FUNCTION_BLOCK "GCS7_E_MYRA_MDEx"	// FB 36
TITLE = MYRA
//
//COPYRIGHT:    (C) 1996 BY  BUHLER LTD.
//                           CH-9240 UZWIL  SWITZERLAND
//
//PRODUCT:      GCS7
//
//TITLE:        MYRA, MYAG, MDEF / MDEA or MDEE 
//              (OPTO22 or 24V signal) 
//
//REVISION:     GCPROVB 11
//-------------------------------------------------------------------------
//
//IDENT:        AUTHOR:             DEPT:                       DATE:
//
//FB36.5.2      A. Egli             CT3                         07-Mar-2007
//              Update Version 5.1 from G. Shingler CDDP
//              - Addition of command 'N' to allow current values to be read
//              - Addition of command 'b' for MYRA to allow current flowrates
//                to be read
//              - Read of average flowrates removed (command 'm')
//FB36.5.1      A. Egli             CT3                         16-Jan-2007
//              - Read average of ingredient 1 to 7 (command i)
//FB36.5.0      G. Shingler         CDDP                        19-Dec-2006
//              - Read actual weights and actual flowrates for feeders
//              - Correction for log alarms
//FB36.4.10     A. Egli             CT3                         25-Sep-2006
//              - Only send commands to the mills that are connected
//FB36.4.9      Ph. Engler          GP92                        03-May-2006
//              - CmdFaultReset set with Gr.CmdFaultReset (M 12.3)
//FB36.4.8      Ph. Engler          GP92                        28-Apr-2006
//              - MDEF: Send 's' only after a 'D'
//              - MDEF: Only one recipe change at the time
//FB36.4.7      A. Egli             CT3                         22-Dec-2004
//              Command 'S': check also MYRA.OutStatus.Suspended
//FB36.4.6      A. Egli             CT3                         05-Nov-2004
//              New transition StFault --> StOn
//FB36.4.5      A. Egli             CT3                         11-Okt-2004
//              Fault reset when InNoMonLC=1
//FB36.4.4      P.Engler            MU664                       20-Sep-2004
//              Condtion for StWaitForResponse --> StOff
//FB36.4.3      A. Egli             CT3                         17-Jun-2004
//              InNoMonLC:No alarm only warning when InpFaultLC
//FB36.4.2      K. Tischer          CT3                         13-JAN-2004
//              Revision=10
//FB36.4.1      A. Egli             CT3                         11-Nov-2002
//              Compare ParAlarmResetTime <0
//FB36.4.0      A. Egli             CT3                         30-Okt-2002
//              Read Actual values of ingredients
//FB36.3.0      A. Egli             CT3                         17-Jun-2002
//              New Release with one block
//              OPTO22 communication to MYRA,MAG and MDEF 
//FB36.2A       A. Egli             CT3                         04-Mai-1998
//              StFault = StCode 32
//FB36.1A       A. Egli             AEE61                       29-Okt-1997
//              1st Release in S7
//
//-------------------------------------------------------------------------
//
//PURPOSE:      MANUAL : see [MYRxxMAN]
//
//              (*1): LC is connected to PC
//                    PLC used 24V signal as interface to PC 
//                   
//                    NOTE: In case of OPTO22 the signal are internal used 
//
//              (*2): LC is connected to PLC by opto22
//
//
//RESTRICTIONS: S7
//              CmdOff, CmdOn: always active unless local mode
//
//-------------------------------------------------------------------------
//=======================================================
//Log Message: 
//------------------------------------------------------
// 0   Off
// 1   On 
// 9   fault cancelled
//10   fault equipement          
//11   fault fault tolerance
//12   fault fault transmision
//
//15   Communcation Fault Opto22
//16   MYAG Alarm
//
//21   MYRA Alarm Hardware
//22   MYRA Alarm Product 
//23   MYRA Alarm Recipe change
//24   MYRA Alarm Feeder 1
//25   MYRA Alarm Feeder 2
//26   MYRA Alarm Feeder 3
//27   MYRA Alarm Feeder 4
//
//41   MDEF Alarm mill 1  
//42   MDEF Alarm mill 2
//43   MDEF Alarm mill 3
//44   MDEF Alarm mill 4
//
//51   MDEF Wrong recipe 1  
//52   MDEF Wrong recipe 2
//53   MDEF Wrong recipe 3  
//54   MDEF Wrong recipe 4  
//
//
//=======================================================
//StCode:  State               
//------------------------------------------------------
//32  StFault                   
// 1  StOff                     
//41  StOff.HWStop                     StOff + InHWStop
//51  StOff.DPFault                    StOff + InDPFault
// 2  StWaitForResponse         
// 3  StOn.Ok                   
// 4  StOn.Warning              
// 5  StCtoFault                
//
AUTHOR : GS
FAMILY : GCS7LL
NAME : MYRA_MDE
VERSION : 5.2
VAR
  StCode : INT ;	//Element state code
  InEnable : BOOL ;	//Enable to run the element
  InDefReady : BOOL ;	//(*1) Answer from PLC: Recipe to sent to MYRA
  InDefFault : BOOL ;	//(*1) Answer from PC:  not eble to send recipe to MYRA
  InNoMonLC : BOOL ;	//No alarm only warning when InpFaultLC
  CmdNewValue : BOOL ;	//Send new target values: Send Flowrate to MYRA
  CmdNewJob : BOOL ;	//Send RecipeNr and Job-Nr to MYRA
  InpOutOfTolerance : BOOL ;	//(*1) Digital input 1=Fault
  InpFaultLc : BOOL ;	//(*1) Digital input 1=HW fault of MYRA
  CmdOff : BOOL ;	//Pulse to stop the element immediately (manual mode)
  CmdOn : BOOL ;	//Pulse to start the element immediately (manual mode)
  CmdNext : BOOL ;	//Pulse to start the element in automatic mode (see global flags)
  CmdFaultReset : BOOL ;	//Command to reset fault
  InLocal : BOOL ;	//1= Local mode (no fault by start with service switch)
  InManual : BOOL ;	//1= Manual/ 0=Automatic
  InReport : BOOL ;	//Report of all state transitions
  spare0307 : BOOL ;
  InHWStop : BOOL ;	//HW stop is detected, no fault
  InDPFault : BOOL ;	//DP-Fault is detected, no fault
  OutWarning : BOOL ;	//Out of tolerance, ParDelayWarning end
  OutDefRequested : BOOL ;	//Definition requested : PC must send recipe to MYRA
  OutComFault : BOOL ;	//Communication vault OPTO22
  OutEnabled : BOOL ;	//Enable to run MYRA (internal used)
  OutpAlarmReset : BOOL ;	//(*1) Digital output: Trigger for alarm reset
  OutpRelease : BOOL ;	//(*1) Digital output: Release measuring
  StOff : BOOL ;	//Element is stopped
  StWaitForResponse : BOOL ;	//PC must send new recipe to MYRA
  StOn : BOOL ;
  StCtoFault : BOOL ;
  StFault : BOOL ;
  MDEF1 : STRUCT 	//OPTO22: MDEF1
   CmdNewRecipe : BOOL ;	//Send recipe to mill
   CmdAlarmReset : BOOL ;	//Send to Mill
   OutSendRecipeNrActive : BOOL ;	//Send of recipe nr is active
   OutSendRecipeNrDone : BOOL ;	//RecipeNr is sent
   OutWrongRecipe : BOOL ;	//Status 4, 6 or 10
   OutAlarm : BOOL ;	//Command 'a'
   StNotOK : BOOL ;
   StOK : BOOL ;
   StFault : BOOL ;
   InRecipeNr : INT ;	//Command 'D'
   Status : INT ;	//Command 's'
  END_STRUCT ;
  MDEF2 : STRUCT 	//OPTO22: MDEF2
   CmdNewRecipe : BOOL ;	//Send recipe to mill
   CmdAlarmReset : BOOL ;	//Send to Mill
   OutSendRecipeNrActive : BOOL ;	//Send of recipe nr is active
   OutSendRecipeNrDone : BOOL ;	//RecipeNr is sent
   OutWrongRecipe : BOOL ;	//Status 4, 6 or 10
   OutAlarm : BOOL ;	//Command 'a'
   StNotOK : BOOL ;
   StOK : BOOL ;
   StFault : BOOL ;
   InRecipeNr : INT ;	//Command 'D'
   Status : INT ;	//Command 's'
  END_STRUCT ;
  MDEF3 : STRUCT 	//OPTO22: MDEF3
   CmdNewRecipe : BOOL ;	//Send recipe to mill
   CmdAlarmReset : BOOL ;	//Send to Mill
   OutSendRecipeNrActive : BOOL ;	//Send of recipe nr is active
   OutSendRecipeNrDone : BOOL ;	//RecipeNr is sent
   OutWrongRecipe : BOOL ;	//Status 4, 6 or 10
   OutAlarm : BOOL ;	//Command 'a'
   StNotOK : BOOL ;
   StOK : BOOL ;
   StFault : BOOL ;
   InRecipeNr : INT ;	//Command 'D'
   Status : INT ;	//Command 's'
  END_STRUCT ;
  MDEF4 : STRUCT 	//OPTO22: MDEF4
   CmdNewRecipe : BOOL ;	//Send recipe to mill
   CmdAlarmReset : BOOL ;	//Send to Mill
   OutSendRecipeNrActive : BOOL ;	//Send of recipe nr is active
   OutSendRecipeNrDone : BOOL ;	//RecipeNr is sent
   OutWrongRecipe : BOOL ;	//Status 4, 6 or 10
   OutAlarm : BOOL ;	//Command 'a'
   StNotOK : BOOL ;
   StOK : BOOL ;
   StFault : BOOL ;
   InRecipeNr : INT ;	//Command 'D'
   Status : INT ;	//Command 's'
  END_STRUCT ;
  MYRA : STRUCT 	//OPTO22: MYRA
   InRecipeNr : INT ;	//Command 'P'
   InJobNr : DINT ;	//Command 'P'
   InFlowrate : DINT ;	//Command 'Q' [kg/h]
   Command : STRUCT 	//Command 'S'
    CheckLimit : BOOL ;
    spare11 : BOOL ;
    spare12 : BOOL ;
    spare13 : BOOL ;
    AlarmReset : BOOL ;	//Is programmed by ASW
    Start : BOOL ;
    spare22 : BOOL ;
    spare23 : BOOL ;
   END_STRUCT ;
   OutAlarm : STRUCT 	//Command 'a'
    SumFault : BOOL ;
    AlarmMYRAHardware : BOOL ;
    AlarmProduct : BOOL ;
    AlarmRecipeChange : BOOL ;
    AlarmFeeder1 : BOOL ;
    AlarmFeeder2 : BOOL ;
    AlarmFeeder3 : BOOL ;
    AlarmFeeder4 : BOOL ;
   END_STRUCT ;
   OutStatus : STRUCT 	//Command 's'
    Started : BOOL ;
    Suspended : BOOL ;
    Remote : BOOL ;
    BatchMode : BOOL ;
    spare4_0 : BOOL ;
    spare4_1 : BOOL ;
    spare4_2 : BOOL ;
    spare4_3 : BOOL ;
    EnableFeeder1 : BOOL ;
    EnableFeeder2 : BOOL ;
    EnableFeeder3 : BOOL ;
    EnableFeeder4 : BOOL ;
    LimitFeeder1 : BOOL ;
    LimitFeeder2 : BOOL ;
    LimitFeeder3 : BOOL ;
    LimitFeeder4 : BOOL ;
   END_STRUCT ;
   OutIngr1 : INT ;	//[1/100%] (Command 'f')
   OutIngr2 : INT ;	//[1/100%] (Command 'f')
   OutIngr3 : INT ;	//[1/100%] (Command 'f')
   OutIngr4 : INT ;	//[1/100%] (Command 'f')
   OutIngr5 : INT ;	//[1/100%] (Command 'f')
   OutIngr6 : INT ;	//[1/100%] (Command 'f')
   OutIngr7 : INT ;	//[1/100%] (Command 'f')
   OutFeeder1Weight : DINT ;	//[5.0] [kg] (Command 'm')
   OutFeeder1Flowrate : DINT ;	//[5.0] [kg/h] (Command 'b')
   OutFeeder2Weight : DINT ;	//[5.0] [kg] (Command 'm')
   OutFeeder2Flowrate : DINT ;	//[5.0] [kg/h] (Command 'b')
   OutFeeder3Weight : DINT ;	//[5.0] [kg] (Command 'm')
   OutFeeder3Flowrate : DINT ;	//[5.0] [kg/h] (Command 'b')
   OutFeeder4Weight : DINT ;	//[5.0] [kg] (Command 'm')
   OutFeeder4Flowrate : DINT ;	//[5.0] [kg/h] (Command 'b')
   OutIngr1Average : INT ;	//[1/100%] (Command 'i')
   OutIngr2Average : INT ;	//[1/100%] (Command 'i')
   OutIngr3Average : INT ;	//[1/100%] (Command 'i')
   OutIngr4Average : INT ;	//[1/100%] (Command 'i')
   OutIngr5Average : INT ;	//[1/100%] (Command 'i')
   OutIngr6Average : INT ;	//[1/100%] (Command 'i')
   OutIngr7Average : INT ;	//[1/100%] (Command 'i')
  END_STRUCT ;
  MYAG : STRUCT 	//OPTO22: MYRG
   Start : BOOL ;	//Command 'I': Is sent to LC (internal used)
   RecipeChange : BOOL ;	//Command 'I': Is sent to LC
   InRecipeNr : INT ;	//ASW: Command 'I': Is sent to LC
   InJobNr : DINT ;	//ASW: Command 'I': Is sent to LC
   OutSumFault : BOOL ;	//Command 'b': Is read from LC
   OutRecipeNr : INT ;	//Command 'b': Is read from LC
   OutJobNr : DINT ;	//Command 'b': Is read from LC
   OutYield1 : INT ;	//Command 'b': Is read from LC
   OutYield2 : INT ;	//Command 'b': Is read from LC
   OutFlowrateAc : DINT ;	//Command 'b': Is read from LC
  END_STRUCT ;
  OutMsg : STRUCT 	//Active Message
   A10LC : BOOL ;
   A11Tolerance : BOOL ;
   A12CommunicationPC : BOOL ;
   A15CommunicationLC : BOOL ;
   A21MYRAHardware : BOOL ;
   A22MYRAProduct : BOOL ;
   A23MYRARecipeChange : BOOL ;
   A24MYRAFeeder1 : BOOL ;
   A25MYRAFeeder2 : BOOL ;
   A26MYRAFeeder3 : BOOL ;
   A27MYRAFeeder4 : BOOL ;
   A41Mill1 : BOOL ;
   A42Mill2 : BOOL ;
   A43Mill3 : BOOL ;
   A44Mill4 : BOOL ;
   A51RecipeMill1 : BOOL ;
   A52RecipeMill3 : BOOL ;
   A53RecipeMill2 : BOOL ;
   A54RecipeMill4 : BOOL ;
  END_STRUCT ;
  OutAlarmNrLog : INT ;	//Last textnumber send to log
  Par : STRUCT
   ParObjectNo : INT ;	//Is used for communication with PC, e.g. for message
   ParMsgType : INT ;	//Is used for message (translation of state)
   ParHornCode : INT ;	//not used
   ParLogOff : BOOL ;	//Report is off
   ParMDEx : BOOL ;	//MDEx: No Delay time if out of tolerance
   ParMYRA : BOOL ;	//OPTO22: MYRA
   ParMDEF : BOOL ;	//OPTO22: MDEF
   ParMYAG : BOOL ;	//OPTO22: MYAG
   ParComDB : INT ;	//OPTO22: Communication DB
   ParLCIdx : INT ;	//OPTO22: Index of data record
   ParLCAddr : INT ;	//OPTO22: Address of LC
   ParNoOfMDEF : INT ;	//OPTO22: Number of connected MDEF
   ParDelayFault : INT ;	//Delay time, until the element changes to fault
   ParAlarmResetTime : INT ;	//Pulse length for OutpFaultReset
   ParResponseTime : INT ;	//Maximum time to wait for answer from PC
   ParDelayWarning : INT ;	//Delay time, until the element changes to StWarning
   OutDelayTime : INT ;	//Actual time
   spare24 : INT ;
   OutHelpFlags : STRUCT 	//Internal used
    OutFaultResetDone : BOOL ;
    OutTestNewAlarm : BOOL ;
    CmdNewValue : BOOL ;
    CmdNewJob : BOOL ;
    OutAlarmActive : BOOL ;
    FlagCheckLimit : BOOL ;
   END_STRUCT ;
   OutComFlags : STRUCT
    a_rDone : BOOL ;
    s_rDone : BOOL ;
    k_Done : BOOL ;
    b_Done : BOOL ;
    D_Done : BOOL ;
    A_Done : BOOL ;
    P_Done : BOOL ;
    Q_Done : BOOL ;
    S_Done : BOOL ;
    I_Done : BOOL ;
    f_rDone : BOOL ;
    m_Done : BOOL ;	//[5.0]
    i_rDone : BOOL ;	//[5.1]
    N_Done : BOOL ;	//[5.2]
   END_STRUCT ;
   OutMillNr : INT ;	//Used for MDEF Telegram
  END_STRUCT ;
END_VAR
VAR_TEMP
  tmpLOGvalue : WORD ;	//LOG value
  tmpLenDyn : DINT ;
  tmpReport : BOOL ;	//Global LOG all
  tmpEnable : BOOL ;	//Global enable
  tmpLocal : BOOL ;
  tmpTimeDone : BOOL ;
  tmpLocalFault : BOOL ;
  tmpOpto22 : BOOL ;
  tmpFBNO : INT ;	//Number of the actual FB
  tmpCommand : INT ;
  tmpComDB : INT ;
  tmpReturn : INT ;
  tmpFault : BOOL ;
  tmpWrongRecipe : BOOL ;
  tmpAddrMsg : DWORD ;
  tmpPar : STRUCT
   ParObjectNo : INT ;	//Is used for communication with PC, e.g. for message
   ParMsgType : INT ;	//Is used for message (translation of state)
   ParHornCode : INT ;	//not used
   ParLogOff : BOOL ;	//Report is off
   ParMDEx : BOOL ;	//MDEx: No Delay time if out of tolerance
   ParMYRA : BOOL ;	//OPTO22: MYRA
   ParMDEF : BOOL ;	//OPTO22: MDEF
   ParMYAG : BOOL ;	//OPTO22: MYAG
   ParComDB : INT ;	//OPTO22: Communication DB
   ParLCIdx : INT ;	//OPTO22: Index of data record
   ParLCAddr : INT ;	//OPTO22: Address of LC
   ParNoOfMDEF : INT ;	//OPTO22: Number of connected MDEF
   ParDelayFault : INT ;	//Delay time, until the element changes to fault
   ParAlarmResetTime : INT ;	//Pulse length for OutpFaultReset
   ParResponseTime : INT ;	//Maximum time to wait for answer from PC
   ParDelayWarning : INT ;	//Delay time, until the element changes to StWarning
   OutMillNr : INT ;	//Used for MDEF Telegram
  END_STRUCT ;
  tmpReturn1 : INT ;
END_VAR
BEGIN
NETWORK
TITLE =  Start Global
      L     170;
      T     #tmpLenDyn;	//--> Len dynamic data in byte
      L     #Par.ParComDB;
      T     #tmpComDB;
      L     36;
      T     #tmpFBNO;
      A     #Par.ParMYRA;
      O     #Par.ParMDEF;
      O     #Par.ParMYAG;
      =     #tmpOpto22;
      TAR2;
      L     DW#16#FFFFFF;
      AD;
      L     P##OutMsg;
      +D;
      T     #tmpAddrMsg;
NETWORK
TITLE =  Call back function (***Opto22***)
////*************************************************
////***             O P T O 22                    ***
////*************************************************
//
//This functions are called by FBxxx (COM) 
      AN    #tmpOpto22;
      JC    PC;
      OPN   DB [#tmpComDB];
      L     0;
      L     DBW 32;	//COM.Element.CODE;
      ==I;
      JC    PC;
//Check if object has moved
      L     #Par.ParObjectNo;
      L     DBD 60;	//COM.LC0.AddrPara;       
      ==D;
      JC    COok;
      BEC;
//=============================================
COok: L     DBB 76;	//COM.Telegram.Command;
      T     #tmpCommand;
      L     1;
      L     DBW 32;	//COM.Element.CODE;
      ==I;
      JC    Send;
      L     2;
      ==I;
      JC    Rcv;
      L     4;	//NAK
      L     DBW 32;	//COM.Element.CODE;
      ==I;
      S     #OutComFault;	//fault MYEB communication
      BEU;
//===== Prepare data for send =================================
//Read telegram length
Send: L     #tmpCommand;
      L     'a';
      ==I;
      AN    #Par.ParMYRA;
      L     4;	//Lenght in byte
      JC    Sndx;
      L     #tmpCommand;
      L     'a';
      ==I;
      A     #Par.ParMYRA;
      L     2;	//Lenght in byte
      JC    Sndx;
      L     #tmpCommand;	//[4.0]
      L     'f';	//[4.0]
      ==I;	//[4.0]
      A     #Par.ParMYRA;	//[4.0]
      L     35;	//Lenght in byte             //[4.0]
      JC    Sndx;
      L     #tmpCommand;	//[5.1]
      L     'i';	//[5.1]
      ==I;	//[5.1]
      A     #Par.ParMYRA;	//[5.1]
      L     28;	//Lenght in byte             //[5.1]
      JC    Sndx;
      L     #tmpCommand;	//[5.0]
      L     'm';	//[5.0]
      ==I;	//[5.0]
      A     #Par.ParMYRA;	//[5.0]
      L     64;	//Lenght in byte //[5.0]
      JC    Sndx;	//[5.0]
      L     #tmpCommand;
      L     's';
      ==I;
      AN    #Par.ParMYRA;
      L     2;	//Lenght in byte
      JC    Sndx;
      L     #tmpCommand;
      L     's';
      ==I;
      A     #Par.ParMYRA;
      L     3;	//Lenght in byte
      JC    Sndx;
      L     #tmpCommand;
      L     'b';	//MYAG
      ==I;
      L     25;	//Lenght in byte
      A     #Par.ParMYAG;	//[5.2]
      JC    Sndx;
      L     #tmpCommand;	//[5.2]
      L     'b';	//[5.2] MYRA
      ==I;	//[5.2]
      L     69;	//[5.2] Lenght in byte
      A     #Par.ParMYRA;	//[5.2]
      JC    Sndx;	//[5.2]
      JU    SndA;
Sndx: T     DBW 86;	//COM.Telegram.LenAnswer
      BEU;
//--------------------
//Send A [3.0]
//--------------------
SndA: L     #tmpCommand;
      L     'A';
      <>I;
      JC    SndD;
// command 1
      L     0;
      T     DBW 40;	//COM.Element.AddrOffset
      L     #Par.OutMillNr;
      T     DBD 36;	//COM.Element.InOutValue
      L     11;	//Convert DInt to 1-ASCII
      T     DBW 0;	//COM.CODE
      CDB;	//ComDB->Instanz-DB
      UC    "GCS7_RS485Ctrl";	//Convert (CODE=DBW0)
      CDB;	//ElementDB->Instanz-DB
      L     1;	//Lenght in byte
      T     DBW 78;	//COM.Telegram.Len
      L     0;	//Lenght in byte
      T     DBW 86;	//COM.Telegram.LenAnswer
      BEU;
//--------------------------
//Send D
//--------------------------
SndD: NOP   0;
      L     #tmpCommand;
      L     'D';
      <>I;
      JC    SndI;
      L     0;	//Character offset
      T     DBW 40;	//COM.Element.AddrOffset
      L     1;
      L     #Par.OutMillNr;
      ==I;
      L     #MDEF1.InRecipeNr;
      JC    SD1;
      L     2;
      L     #Par.OutMillNr;
      ==I;
      L     #MDEF2.InRecipeNr;
      JC    SD1;
      L     3;
      L     #Par.OutMillNr;
      ==I;
      L     #MDEF3.InRecipeNr;
      JC    SD1;
      L     #MDEF4.InRecipeNr;
SD1:  T     DBD 36;	//COM.Element.InOutValue
      L     13;	//Convert DInt to 3-ASCII
      T     DBW 0;	//COM.CODE
      CDB;	//ComDB->Instanz-DB
      UC    "GCS7_RS485Ctrl";	//Convert (CODE=DBW0)
      CDB;	//ElementDB->Instanz-DB
      L     3;	//Lenght in byte
      T     DBW 78;	//COM.Telegram.Len
      L     0;	//Lenght in byte
      T     DBW 86;	//COM.Telegram.LenAnswer
      BEU;
//--------------------------
//Send I
//--------------------------
SndI: NOP   0;
      L     #tmpCommand;
      L     'I';
      <>I;
//[5.2]      JC    SndP
      JC    SndN;	//[5.2]
//Start
      L     0;	//Character offset
      T     DBW 40;	//COM.Element.AddrOffset
      L     0;
      T     DBD 36;	//COM.Element.InOutValue
      A     #MYAG.Start;
      =     DBX 39.0;
      L     11;	//Convert DInt to 1-ASCII
      T     DBW 0;	//COM.CODE
      CDB;	//ComDB->Instanz-DB
      UC    "GCS7_RS485Ctrl";	//Convert (CODE=DBW0)
      CDB;	//ElementDB->Instanz-DB
//Recipe change
      L     1;	//Character offset
      T     DBW 40;	//COM.Element.AddrOffset
      L     0;
      T     DBD 36;	//COM.Element.InOutValue
      A     #InManual;
      ON    #InLocal;
      AN    #InDefReady;
      =     #MYAG.RecipeChange;
      =     DBX 39.0;
      L     11;	//Convert DInt to 1-ASCII
      T     DBW 0;	//COM.CODE
      CDB;	//ComDB->Instanz-DB
      UC    "GCS7_RS485Ctrl";	//Convert (CODE=DBW0)
      CDB;	//ElementDB->Instanz-DB
//RecipeNr
      L     2;	//Character offset
      T     DBW 40;	//COM.Element.AddrOffset
      L     #MYAG.InRecipeNr;
      T     DBD 36;	//COM.Element.InOutValue
      L     12;	//Convert DInt to 1-ASCII
      T     DBW 0;	//COM.CODE
      CDB;	//ComDB->Instanz-DB
      UC    "GCS7_RS485Ctrl";	//Convert (CODE=DBW0)
      CDB;	//ElementDB->Instanz-DB
//JobNr
      L     4;	//Character offset
      T     DBW 40;	//COM.Element.AddrOffset
      L     #MYAG.InJobNr;
      T     DBD 36;	//COM.Element.InOutValue
      T     DBD 36;	//COM.Element.InOutValue
      L     16;	//Convert DInt to 1-ASCII
      T     DBW 0;	//COM.CODE
      CDB;	//ComDB->Instanz-DB
      UC    "GCS7_RS485Ctrl";	//Convert (CODE=DBW0)
      CDB;	//ElementDB->Instanz-DB
      L     10;	//Lenght in byte
      T     DBW 78;	//COM.Telegram.Len
      L     0;	//Lenght in byte
      T     DBW 86;	//COM.Telegram.LenAnswer
      BEU;
//[5.2]--------------------------
//[5.2]Send N
//[5.2]--------------------------
SndN: L     #tmpCommand;	//[5.2]
      L     'N';	//[5.2]
      <>I;	//[5.2]
      JC    SndP;	//[5.2]
//[5.2] Job reference 
      L     0;	//[5.2]Character offset
      T     DBW 40;	//[5.2]COM.Element.AddrOffset
      L     0;	//[5.2]0 =  current job
      T     DBD 36;	//[5.2]COM.Element.InOutValue
      L     16;	//[5.2]Convert DInt to 6-ASCII
      T     DBW 0;	//[5.2]COM.CODE
      CDB;	//[5.2]ComDB->Instanz-DB
      UC    "GCS7_RS485Ctrl";	//[5.2]Convert (CODE=DBW0)
      CDB;	//[5.2]ElementDB->Instanz-DB
      L     6;	//[5.2]Lenght in byte
      T     DBW 78;	//[5.2]COM.Telegram.Len
      L     0;	//[5.2]Lenght in byte
      T     DBW 86;	//[5.2]COM.Telegram.LenAnswer
      BEU;
//--------------------------
//Send P
//--------------------------
SndP: L     #tmpCommand;
      L     'P';
      <>I;
      JC    SndQ;
//RecipeNr 
      L     0;	//Character offset
      T     DBW 40;	//COM.Element.AddrOffset
      L     #MYRA.InRecipeNr;
      T     DBD 36;	//COM.Element.InOutValue
      L     13;	//Convert DInt to 3-ASCII
      T     DBW 0;	//COM.CODE
      CDB;	//ComDB->Instanz-DB
      UC    "GCS7_RS485Ctrl";	//Convert (CODE=DBW0)
      CDB;	//ElementDB->Instanz-DB
//Order Number
      L     3;	//Character offset
      T     DBW 40;	//COM.Element.AddrOffset
      L     #MYRA.InJobNr;
      T     DBD 36;	//COM.Element.InOutValue
      L     16;	//Convert DInt to 6-ASCII
      T     DBW 0;	//COM.CODE
      CDB;	//ComDB->Instanz-DB
      UC    "GCS7_RS485Ctrl";	//Convert (CODE=DBW0)
      CDB;	//ElementDB->Instanz-DB
      L     9;	//Lenght in byte
      T     DBW 78;	//COM.Telegram.Len
      L     0;	//Lenght in byte
      T     DBW 86;	//COM.Telegram.LenAnswer
      BEU;
//--------------------------
//Send Q
//--------------------------
SndQ: L     #tmpCommand;
      L     'Q';
      <>I;
      JC    SndS;
//Flowrate
      L     0;	//Character offset
      T     DBW 40;	//COM.Element.AddrOffset
      L     #MYRA.InFlowrate;
      T     DBD 36;	//COM.Element.InOutValue
      L     16;	//Convert DInt to 6-ASCII
      T     DBW 0;	//COM.CODE
      CDB;	//ComDB->Instanz-DB
      UC    "GCS7_RS485Ctrl";	//Convert (CODE=DBW0)
      CDB;	//ElementDB->Instanz-DB
      L     6;	//Lenght in byte
      T     DBW 78;	//COM.Telegram.Len
      L     0;	//Lenght in byte
      T     DBW 86;	//COM.Telegram.LenAnswer
      BEU;
//--------------------------
//Send S
//--------------------------
SndS: L     #tmpCommand;
      L     'S';
      <>I;
      JC    SndZ;
      A     #MYRA.Command.AlarmReset;
      S     #Par.OutHelpFlags.OutFaultResetDone;
//Start
      L     0;	//Character offset
      T     DBW 40;	//COM.Element.AddrOffset
      L     0;
      T     DBD 36;	//COM.Element.InOutValue
      CALL  "SIEMENS_BLKMOV" (
           SRCBLK                   := #MYRA.Command,
           RET_VAL                  := #tmpReturn,
           DSTBLK                   := DBB 39);
      L     32;	//Convert Hex to 2-ASCII
      T     DBW 0;	//COM.CODE
      CDB;	//ComDB->Instanz-DB
      UC    "GCS7_RS485Ctrl";	//Convert (CODE=DBW0)
      CDB;	//ElementDB->Instanz-DB
      L     2;	//Lenght in byte
      T     DBW 78;	//COM.Telegram.Len
      L     0;	//Lenght in byte
      T     DBW 86;	//COM.Telegram.LenAnswer
      BEU;
SndZ: BEU;
//--- Get done ---------------
//Copy reveived data to element
//--------------------------
//Receive f [4.]
//--------------------------
Rcv:  R     #OutComFault;
      L     #tmpCommand;
      L     'f';
      <>I;
      JC    Rcvi;
//OutIngr1 
      L     0;	//Character offset
      T     DBW 40;	//COM.Element.AddrOffset
      L     25;	//Convert 5-ASCII to DInt
      T     DBW 0;	//COM.CODE
      CDB;	//ComDB->Instanz-DB
      UC    "GCS7_RS485Ctrl";	//Convert (CODE=DBW0)
      CDB;	//ElementDB->Instanz-DB
      L     DBD 36;	//COM.Element.InOutValue
      DTR;
      L     1.000001e-01;
      *R;
      RND;
      T     #MYRA.OutIngr1;
//OutIngr2
      L     5;	//Character offset
      T     DBW 40;	//COM.Element.AddrOffset
      L     25;	//Convert 5-ASCII to DInt
      T     DBW 0;	//COM.CODE
      CDB;	//ComDB->Instanz-DB
      UC    "GCS7_RS485Ctrl";	//Convert (CODE=DBW0)
      CDB;	//ElementDB->Instanz-DB
      L     DBD 36;	//COM.Element.InOutValue
      DTR;
      L     1.000001e-01;
      *R;
      RND;
      T     #MYRA.OutIngr2;
//OutIngr3
      L     10;	//Character offset
      T     DBW 40;	//COM.Element.AddrOffset
      L     25;	//Convert 5-ASCII to DInt
      T     DBW 0;	//COM.CODE
      CDB;	//ComDB->Instanz-DB
      UC    "GCS7_RS485Ctrl";	//Convert (CODE=DBW0)
      CDB;	//ElementDB->Instanz-DB
      L     DBD 36;	//COM.Element.InOutValue
      DTR;
      L     1.000001e-01;
      *R;
      RND;
      T     #MYRA.OutIngr3;
//OutIngr4
      L     15;	//Character offset
      T     DBW 40;	//COM.Element.AddrOffset
      L     25;	//Convert 5-ASCII to DInt
      T     DBW 0;	//COM.CODE
      CDB;	//ComDB->Instanz-DB
      UC    "GCS7_RS485Ctrl";	//Convert (CODE=DBW0)
      CDB;	//ElementDB->Instanz-DB
      L     DBD 36;	//COM.Element.InOutValue
      DTR;
      L     1.000001e-01;
      *R;
      RND;
      T     #MYRA.OutIngr4;
//OutIngr5
      L     20;	//Character offset
      T     DBW 40;	//COM.Element.AddrOffset
      L     25;	//Convert 5-ASCII to DInt
      T     DBW 0;	//COM.CODE
      CDB;	//ComDB->Instanz-DB
      UC    "GCS7_RS485Ctrl";	//Convert (CODE=DBW0)
      CDB;	//ElementDB->Instanz-DB
      L     DBD 36;	//COM.Element.InOutValue
      DTR;
      L     1.000001e-01;
      *R;
      RND;
      T     #MYRA.OutIngr5;
//OutIngr6
      L     25;	//Character offset
      T     DBW 40;	//COM.Element.AddrOffset
      L     25;	//Convert 5-ASCII to DInt
      T     DBW 0;	//COM.CODE
      CDB;	//ComDB->Instanz-DB
      UC    "GCS7_RS485Ctrl";	//Convert (CODE=DBW0)
      CDB;	//ElementDB->Instanz-DB
      L     DBD 36;	//COM.Element.InOutValue
      DTR;
      L     1.000001e-01;
      *R;
      RND;
      T     #MYRA.OutIngr6;
//OutIngr7
      L     30;	//Character offset
      T     DBW 40;	//COM.Element.AddrOffset
      L     25;	//Convert 5-ASCII to DInt
      T     DBW 0;	//COM.CODE
      CDB;	//ComDB->Instanz-DB
      UC    "GCS7_RS485Ctrl";	//Convert (CODE=DBW0)
      CDB;	//ElementDB->Instanz-DB
      L     DBD 36;	//COM.Element.InOutValue
      DTR;
      L     1.000001e-01;
      *R;
      RND;
      T     #MYRA.OutIngr7;
      BEU;
//--------------------------
//Receive i
//--------------------------
//[5.1]--->
Rcvi: L     #tmpCommand;
      L     'i';
      <>I;
      JC    Rcva;
//OutIngr1 
      L     0;	//Character offset
      T     DBW 40;	//COM.Element.AddrOffset
      L     24;	//Convert 4-ASCII to DInt
      T     DBW 0;	//COM.CODE
      CDB;	//ComDB->Instanz-DB
      UC    "GCS7_RS485Ctrl";	//Convert (CODE=DBW0)
      CDB;	//ElementDB->Instanz-DB
      L     DBD 36;	//COM.Element.InOutValue
      T     #MYRA.OutIngr1Average;
//OutIngr2
      L     4;	//Character offset
      T     DBW 40;	//COM.Element.AddrOffset
      L     24;	//Convert 4-ASCII to DInt
      T     DBW 0;	//COM.CODE
      CDB;	//ComDB->Instanz-DB
      UC    "GCS7_RS485Ctrl";	//Convert (CODE=DBW0)
      CDB;	//ElementDB->Instanz-DB
      L     DBD 36;	//COM.Element.InOutValue
      T     #MYRA.OutIngr2Average;
//OutIngr3
      L     8;	//Character offset
      T     DBW 40;	//COM.Element.AddrOffset
      L     24;	//Convert 4-ASCII to DInt
      T     DBW 0;	//COM.CODE
      CDB;	//ComDB->Instanz-DB
      UC    "GCS7_RS485Ctrl";	//Convert (CODE=DBW0)
      CDB;	//ElementDB->Instanz-DB
      L     DBD 36;	//COM.Element.InOutValue
      T     #MYRA.OutIngr3Average;
//OutIngr4
      L     12;	//Character offset
      T     DBW 40;	//COM.Element.AddrOffset
      L     24;	//Convert 4-ASCII to DInt
      T     DBW 0;	//COM.CODE
      CDB;	//ComDB->Instanz-DB
      UC    "GCS7_RS485Ctrl";	//Convert (CODE=DBW0)
      CDB;	//ElementDB->Instanz-DB
      L     DBD 36;	//COM.Element.InOutValue
      T     #MYRA.OutIngr4Average;
//OutIngr5
      L     16;	//Character offset
      T     DBW 40;	//COM.Element.AddrOffset
      L     24;	//Convert 4-ASCII to DInt
      T     DBW 0;	//COM.CODE
      CDB;	//ComDB->Instanz-DB
      UC    "GCS7_RS485Ctrl";	//Convert (CODE=DBW0)
      CDB;	//ElementDB->Instanz-DB
      L     DBD 36;	//COM.Element.InOutValue
      T     #MYRA.OutIngr5Average;
//OutIngr6
      L     20;	//Character offset
      T     DBW 40;	//COM.Element.AddrOffset
      L     24;	//Convert 4-ASCII to DInt
      T     DBW 0;	//COM.CODE
      CDB;	//ComDB->Instanz-DB
      UC    "GCS7_RS485Ctrl";	//Convert (CODE=DBW0)
      CDB;	//ElementDB->Instanz-DB
      L     DBD 36;	//COM.Element.InOutValue
      T     #MYRA.OutIngr6Average;
//OutIngr7
      L     24;	//Character offset
      T     DBW 40;	//COM.Element.AddrOffset
      L     24;	//Convert 4-ASCII to DInt
      T     DBW 0;	//COM.CODE
      CDB;	//ComDB->Instanz-DB
      UC    "GCS7_RS485Ctrl";	//Convert (CODE=DBW0)
      CDB;	//ElementDB->Instanz-DB
      L     DBD 36;	//COM.Element.InOutValue
      T     #MYRA.OutIngr7Average;
      BEU;
//<---[5.1]
//--------------------------
//Receive a
//--------------------------
Rcva: L     #tmpCommand;
      L     'a';
      <>I;
      JC    Rcvs;
      A     #Par.OutHelpFlags.OutFaultResetDone;
      R     #Par.OutHelpFlags.OutFaultResetDone;
      S     #Par.OutHelpFlags.OutTestNewAlarm;
      AN    #Par.ParMYRA;
      JC    aMDF;
//--------------------------
//Receive 'a' MYRA
//--------------------------
//OutAlarmNrMill1
      L     0;	//Character offset
      T     DBW 40;	//COM.Element.AddrOffset
      L     42;	//Convert 1-ASCII to Hex
      T     DBW 0;	//COM.CODE
      CDB;	//ComDB->Instanz-DB
      UC    "GCS7_RS485Ctrl";	//Convert (CODE=DBW0)
      CDB;	//ElementDB->Instanz-DB
      CALL  "SIEMENS_BLKMOV" (
           SRCBLK                   := DBB 39,
           RET_VAL                  := #tmpReturn,
           DSTBLK                   := #MYRA.OutAlarm);
      BEU;
//--------------------------
//Receive 'a' MDEF
//--------------------------
//OutAlarmNrMill1
aMDF: L     0;	//Character offset
      T     DBW 40;	//COM.Element.AddrOffset
      L     41;	//Convert 1-ASCII to Hex
      T     DBW 0;	//COM.CODE
      CDB;	//ComDB->Instanz-DB
      UC    "GCS7_RS485Ctrl";	//Convert (CODE=DBW0)
      CDB;	//ElementDB->Instanz-DB
      L     DBD 36;	//COM.Element.InOutValue
      L     1;
      ==I;
      =     #MDEF1.OutAlarm;
//OutAlarmNrMill2
      L     1;	//Character offset
      T     DBW 40;	//COM.Element.AddrOffset
      L     41;	//Convert 1-ASCII to Hex
      T     DBW 0;	//COM.CODE
      CDB;	//ComDB->Instanz-DB
      UC    "GCS7_RS485Ctrl";	//Convert (CODE=DBW0)
      CDB;	//ElementDB->Instanz-DB
      L     DBD 36;	//COM.Element.InOutValue
      L     1;
      ==I;
      =     #MDEF2.OutAlarm;
//OutAlarmNrMill3
      L     2;	//Character offset
      T     DBW 40;	//COM.Element.AddrOffset
      L     41;	//Convert 1-ASCII to Hex
      T     DBW 0;	//COM.CODE
      CDB;	//ComDB->Instanz-DB
      UC    "GCS7_RS485Ctrl";	//Convert (CODE=DBW0)
      CDB;	//ElementDB->Instanz-DB
      L     DBD 36;	//COM.Element.InOutValue
      L     1;
      ==I;
      =     #MDEF3.OutAlarm;
//OutAlarmNrMill4
      L     3;	//Character offset
      T     DBW 40;	//COM.Element.AddrOffset
      L     41;	//Convert 1-ASCII to Hex
      T     DBW 0;	//COM.CODE
      CDB;	//ComDB->Instanz-DB
      UC    "GCS7_RS485Ctrl";	//Convert (CODE=DBW0)
      CDB;	//ElementDB->Instanz-DB
      L     DBD 36;	//COM.Element.InOutValue
      L     1;
      ==I;
      =     #MDEF4.OutAlarm;
      BEU;
//--------------------------
//Receive s
//--------------------------
Rcvs: L     #tmpCommand;
      L     's';
      <>I;
      JC    Rcvb;
      AN    #Par.ParMYRA;
      JC    sMDF;
//--------------------------
//Receive 's' MYRA
//--------------------------
      L     0;	//Character offset
      T     DBW 40;	//COM.Element.AddrOffset
      L     43;	//Convert 1-ASCII to Hex
      T     DBW 0;	//COM.CODE
      CDB;	//ComDB->Instanz-DB
      UC    "GCS7_RS485Ctrl";	//Convert (CODE=DBW0)
      CDB;	//ElementDB->Instanz-DB
      CALL  "SIEMENS_BLKMOV" (
           SRCBLK                   := DBW 38,
           RET_VAL                  := #tmpReturn,
           DSTBLK                   := #MYRA.OutStatus);
      BEU;
//--------------------------
//Receive 's' MDEF
//--------------------------
sMDF: L     0;	//Character offset
      T     DBW 40;	//COM.Element.AddrOffset
      L     22;	//Convert 2-ASCII to DInt
      T     DBW 0;	//COM.CODE
      CDB;	//ComDB->Instanz-DB
      UC    "GCS7_RS485Ctrl";	//Convert (CODE=DBW0)
      CDB;	//ElementDB->Instanz-DB
      L     4;
      L     DBD 36;	//COM.Element.InOutValue
      ==I;
      O(;
      L     6;	//[4.8]
      ==I;
      );
      O(;
      L     10;
      L     DBD 36;	//COM.Element.InOutValue
      ==I;
      );
      =     #tmpWrongRecipe;
      L     #Par.OutMillNr;
      L     1;
      <>I;
      JC    sM2;
      L     DBD 36;	//COM.Element.InOutValue
      T     #MDEF1.Status;
      L     0;
      ==I;
      A     #MDEF1.OutSendRecipeNrActive;
      S     #MDEF1.OutSendRecipeNrDone;
//[4.8]      R     #MDEF1.CmdNewRecipe
      SET;
      R     #MDEF1.CmdNewRecipe;	//[4.8]
      R     #MDEF1.OutSendRecipeNrActive;
      A     #tmpWrongRecipe;
      =     #MDEF1.OutWrongRecipe;
      BEU;
sM2:  L     #Par.OutMillNr;
      L     2;
      <>I;
      JC    sM3;
      L     DBD 36;	//COM.Element.InOutValue
      T     #MDEF2.Status;
      L     0;
      ==I;
      A     #MDEF2.OutSendRecipeNrActive;
      S     #MDEF2.OutSendRecipeNrDone;
//[4.8]      R     #MDEF2.CmdNewRecipe
      SET;
      R     #MDEF2.CmdNewRecipe;	//[4.8]
      R     #MDEF2.OutSendRecipeNrActive;
      A     #tmpWrongRecipe;
      =     #MDEF2.OutWrongRecipe;
      BEU;
sM3:  L     #Par.OutMillNr;
      L     3;
      <>I;
      JC    sM4;
      L     DBD 36;	//COM.Element.InOutValue
      T     #MDEF3.Status;
      L     0;
      ==I;
      A     #MDEF3.OutSendRecipeNrActive;
      S     #MDEF3.OutSendRecipeNrDone;
//[4.8]      R     #MDEF3.CmdNewRecipe
      SET;
      R     #MDEF3.CmdNewRecipe;	//[4.8]
      R     #MDEF3.OutSendRecipeNrActive;
      A     #tmpWrongRecipe;
      =     #MDEF3.OutWrongRecipe;
      BEU;
sM4:  L     DBD 36;	//COM.Element.InOutValue
      T     #MDEF4.Status;
      L     0;
      ==I;
      A     #MDEF4.OutSendRecipeNrActive;
      S     #MDEF4.OutSendRecipeNrDone;
//[4.8]      R     #MDEF4.CmdNewRecipe
      SET;
      R     #MDEF4.CmdNewRecipe;	//[4.8]
      R     #MDEF4.OutSendRecipeNrActive;
      A     #tmpWrongRecipe;
      =     #MDEF4.OutWrongRecipe;
      BEU;
//--------------------------
//Receive b
//--------------------------
Rcvb: L     #tmpCommand;
      L     'b';
      <>I;
// [5.0]      JC    RcvP; 
      JC    Rcvm;	// [5.0]
      A     #Par.ParMYRA;	//[5.2]
      JC    bMYR;	//[5.2]
//--------------------------
//Receive b MYAG
//--------------------------
//Alarm
      L     0;	//Character offset
      T     DBW 40;	//COM.Element.AddrOffset
      L     41;	//Convert 1-ASCII to Hex
      T     DBW 0;	//COM.CODE
      CDB;	//ComDB->Instanz-DB
      UC    "GCS7_RS485Ctrl";	//Convert (CODE=DBW0)
      CDB;	//ElementDB->Instanz-DB
      A     DBX 39.0;	//COM.Element.InOutValue
      =     #MYAG.OutSumFault;
//AlarmRecipe  
      L     1;	//Character offset
      T     DBW 40;	//COM.Element.AddrOffset
      L     22;	//Convert 2-ASCII to DInt
      T     DBW 0;	//COM.CODE
      CDB;	//ComDB->Instanz-DB
      UC    "GCS7_RS485Ctrl";	//Convert (CODE=DBW0)
      CDB;	//ElementDB->Instanz-DB
      L     DBD 36;	//COM.Element.InOutValue
      T     #MYAG.OutRecipeNr;
//JobNr  
      L     3;	//Character offset
      T     DBW 40;	//COM.Element.AddrOffset
      L     26;	//Convert 2-ASCII to DInt
      T     DBW 0;	//COM.CODE
      CDB;	//ComDB->Instanz-DB
      UC    "GCS7_RS485Ctrl";	//Convert (CODE=DBW0)
      CDB;	//ElementDB->Instanz-DB
      L     DBD 36;	//COM.Element.InOutValue
      T     #MYAG.OutJobNr;
//Yield1  
      L     9;	//Character offset
      T     DBW 40;	//COM.Element.AddrOffset
      L     24;	//Convert 2-ASCII to DInt
      T     DBW 0;	//COM.CODE
      CDB;	//ComDB->Instanz-DB
      UC    "GCS7_RS485Ctrl";	//Convert (CODE=DBW0)
      CDB;	//ElementDB->Instanz-DB
      L     DBD 36;	//COM.Element.InOutValue
      T     #MYAG.OutYield1;
//Yield2  
      L     13;	//Character offset
      T     DBW 40;	//COM.Element.AddrOffset
      L     24;	//Convert 2-ASCII to DInt
      T     DBW 0;	//COM.CODE
      CDB;	//ComDB->Instanz-DB
      UC    "GCS7_RS485Ctrl";	//Convert (CODE=DBW0)
      CDB;	//ElementDB->Instanz-DB
      L     DBD 36;	//COM.Element.InOutValue
      T     #MYAG.OutYield2;
//Yield2  
      L     17;	//Character offset
      T     DBW 40;	//COM.Element.AddrOffset
      L     28;	//Convert 2-ASCII to DInt
      T     DBW 0;	//COM.CODE
      CDB;	//ComDB->Instanz-DB
      UC    "GCS7_RS485Ctrl";	//Convert (CODE=DBW0)
      CDB;	//ElementDB->Instanz-DB
      L     DBD 36;	//COM.Element.InOutValue
      T     #MYAG.OutFlowrateAc;
      BEU;
//[5.2]--------------------------
//[5.2]Receive b MYRA
//[5.2]--------------------------
bMYR: NOP   0;	//[5.2]
//[5.2] OutFeeder1 flowrate
      L     37;	//[5.2] Character offset
      T     DBW 40;	//[5.2] COM.Element.AddrOffset
      L     28;	//[5.2] Convert 8-ASCII to DInt
      T     DBW 0;	//[5.2] COM.CODE
      CDB;	//[5.2] ComDB->Instanz-DB
      UC    "GCS7_RS485Ctrl";	//[5.2] Convert (CODE=DBW0)
      CDB;	//[5.2] ElementDB->Instanz-DB
      L     DBD 36;	//[5.2] COM.Element.InOutValue
      T     #MYRA.OutFeeder1Flowrate;	//[5.2]
//[5.2] OutFeeder2 flowrate
      L     45;	//[5.2] Character offset
      T     DBW 40;	//[5.2] COM.Element.AddrOffset
      L     28;	//[5.2] Convert 8-ASCII to DInt
      T     DBW 0;	//[5.2] COM.CODE
      CDB;	//[5.2] ComDB->Instanz-DB
      UC    "GCS7_RS485Ctrl";	//[5.2] Convert (CODE=DBW0)
      CDB;	//[5.2] ElementDB->Instanz-DB
      L     DBD 36;	//[5.2] COM.Element.InOutValue
      T     #MYRA.OutFeeder2Flowrate;	//[5.2]
//[5.2] OutFeeder3 flowrate
      L     53;	//[5.2] Character offset
      T     DBW 40;	//[5.2] COM.Element.AddrOffset
      L     28;	//[5.2] Convert 8-ASCII to DInt
      T     DBW 0;	//[5.2] COM.CODE
      CDB;	//[5.2] ComDB->Instanz-DB
      UC    "GCS7_RS485Ctrl";	//[5.2] Convert (CODE=DBW0)
      CDB;	//[5.2] ElementDB->Instanz-DB
      L     DBD 36;	//[5.2] COM.Element.InOutValue
      T     #MYRA.OutFeeder3Flowrate;	//[5.2]
//[5.2] OutFeeder4 flowrate
      L     61;	//[5.2] Character offset
      T     DBW 40;	//[5.2] COM.Element.AddrOffset
      L     28;	//[5.2] Convert 8-ASCII to DInt
      T     DBW 0;	//[5.2] COM.CODE
      CDB;	//[5.2] ComDB->Instanz-DB
      UC    "GCS7_RS485Ctrl";	//[5.2] Convert (CODE=DBW0)
      CDB;	//[5.2] ElementDB->Instanz-DB
      L     DBD 36;	//[5.2] COM.Element.InOutValue
      T     #MYRA.OutFeeder4Flowrate;	//[5.2]
      BEU;	//[5.2]
//--------------------------
//Receive m [5.0]
//--------------------------
Rcvm: L     #tmpCommand;	//[5.0]
      L     'm';	//[5.0]
      <>I;	//[5.0]
      JC    RcvP;	//[5.0]
//[5.0] OutFeeder1 weight
      L     0;	//[5.0] Character offset
      T     DBW 40;	//[5.0] COM.Element.AddrOffset
      L     28;	//[5.0] Convert 8-ASCII to DInt
      T     DBW 0;	//[5.0] COM.CODE
      CDB;	//[5.0] ComDB->Instanz-DB
      UC    "GCS7_RS485Ctrl";	//[5.0] Convert (CODE=DBW0)
      CDB;	//[5.0] ElementDB->Instanz-DB
      L     DBD 36;	//[5.0] COM.Element.InOutValue
      T     #MYRA.OutFeeder1Weight;	//[5.0]
//[5.0] OutFeeder2 weight
      L     8;	//[5.0] Character offset
      T     DBW 40;	//[5.0] COM.Element.AddrOffset
      L     28;	//[5.0] Convert 8-ASCII to DInt
      T     DBW 0;	//[5.0] COM.CODE
      CDB;	//[5.0] ComDB->Instanz-DB
      UC    "GCS7_RS485Ctrl";	//[5.0] Convert (CODE=DBW0)
      CDB;	//[5.0] ElementDB->Instanz-DB
      L     DBD 36;	//[5.0] COM.Element.InOutValue
      T     #MYRA.OutFeeder2Weight;	//[5.0]
//[5.0] OutFeeder3 weight
      L     16;	//[5.0] Character offset
      T     DBW 40;	//[5.0] COM.Element.AddrOffset
      L     28;	//[5.0] Convert 8-ASCII to DInt
      T     DBW 0;	//[5.0] COM.CODE
      CDB;	//[5.0] ComDB->Instanz-DB
      UC    "GCS7_RS485Ctrl";	//[5.0] Convert (CODE=DBW0)
      CDB;	//[5.0] ElementDB->Instanz-DB
      L     DBD 36;	//[5.0] COM.Element.InOutValue
      T     #MYRA.OutFeeder3Weight;	//[5.0]
//[5.0] OutFeeder4 weight
      L     24;	//[5.0] Character offset
      T     DBW 40;	//[5.0] COM.Element.AddrOffset
      L     28;	//[5.0] Convert 8-ASCII to DInt
      T     DBW 0;	//[5.0] COM.CODE
      CDB;	//[5.0] ComDB->Instanz-DB
      UC    "GCS7_RS485Ctrl";	//[5.0] Convert (CODE=DBW0)
      CDB;	//[5.0] ElementDB->Instanz-DB
      L     DBD 36;	//[5.0] COM.Element.InOutValue
      T     #MYRA.OutFeeder4Weight;	//[5.0]
      BEU;	//[5.0]
//--------------------------
//Receive P
//--------------------------
RcvP: L     #tmpCommand;
      L     'P';
      <>I;
      JC    RcvQ;
      S     #Par.OutComFlags.P_Done;
      R     #Par.OutHelpFlags.CmdNewJob;
      BEU;
//--------------------------
//Receive Q
//--------------------------
RcvQ: L     #tmpCommand;
      L     'Q';
      <>I;
      JC    RcvS;
      S     #Par.OutComFlags.Q_Done;
      R     #Par.OutHelpFlags.CmdNewValue;
      BEU;
//--------------------------
//Receive S
//--------------------------
RcvS: L     #tmpCommand;
      L     'S';
      <>I;
      JC    RcvI;
      S     #Par.OutComFlags.S_Done;
      A     #MYRA.Command.CheckLimit;
      =     #Par.OutHelpFlags.FlagCheckLimit;
      A     #MYRA.Command.AlarmReset;
      R     #MYRA.Command.AlarmReset;
      BEU;
//--------------------------
//Receive I
//--------------------------
RcvI: L     #tmpCommand;
      L     'I';
      <>I;
      JC    RcvD;
      S     #Par.OutComFlags.I_Done;
      BEU;
//--------------------------
//Receive D
//--------------------------
RcvD: L     #tmpCommand;
      L     'D';
      <>I;
      JC    RcvA;
      S     #Par.OutComFlags.D_Done;
      L     #Par.OutMillNr;
      L     1;
      ==I;
      S     #MDEF1.OutSendRecipeNrActive;
      L     #Par.OutMillNr;
      L     2;
      ==I;
      S     #MDEF2.OutSendRecipeNrActive;
      L     #Par.OutMillNr;
      L     3;
      ==I;
      S     #MDEF3.OutSendRecipeNrActive;
      L     #Par.OutMillNr;
      L     4;
      ==I;
      S     #MDEF4.OutSendRecipeNrActive;
      BEU;
//--------------------------
//Receive A
//--------------------------
RcvA: L     #tmpCommand;
      L     'A';
      <>I;
      JC    RcvZ;
      S     #Par.OutComFlags.A_Done;
      S     #Par.OutHelpFlags.OutFaultResetDone;
      BEU;
RcvZ: BEU;
PC:   NOP   0;
NETWORK
TITLE = PC Control
//=== Test Object number =====================
      L     "SYS_DirectCtrlDB".PC.ObjectNo;	//PCControl.ObjectNo
      L     #Par.ParObjectNo;	//Input ObjectNo
      <>I;
      JC    Ctrl;
//===     Test OType      ========================
      L     1036;	//Input object type
      L     "SYS_DirectCtrlDB".PC.ObjectType;	//PCControl.ObjectType
      <>I;
      JC    Ctrl;
//=== Test Handshake =========================
      A     "SYS_DirectCtrlDB".PC.Hsk.FExamine;	// Handshake.FExamine
      JC    pExa;
      A     "SYS_DirectCtrlDB".PC.Hsk.FDefineCmd;	// Handshake.FDefineCmd
      JC    pCmd;
      A     "SYS_DirectCtrlDB".PC.Hsk.FDefinePara;	// Handshake.FDefinePara
      JC    pPar;
pIni: L     2;	// FcInit
      UC    "SYS_DirectCtrl";
      JU    Ctrl;
// Write parameter 
pPar: LAR1  P#DBX 58.0;
      L     P##Par;
      L     DW#16#FFFFF;
      AD;
      +AR1;
      L     DBW [AR1,P#16.0];
      T     #Par.ParDelayFault;
      L     DBW [AR1,P#18.0];
      T     #Par.ParAlarmResetTime;
      L     DBW [AR1,P#20.0];
      T     #Par.ParResponseTime;
      L     DBW [AR1,P#22.0];
      T     #Par.ParDelayWarning;
// Write new commands from PC to Interface object
pCmd: A     "SYS_DirectCtrlDB".PC.Cmd1[8];	// CmdOff
      S     #CmdOff;
      A     "SYS_DirectCtrlDB".PC.Cmd1[9];	// CmdOn
      S     #CmdOn;
      A     "SYS_DirectCtrlDB".PC.Cmd1[10];	// CmdNext
      S     #CmdNext;
      A     "SYS_DirectCtrlDB".PC.Cmd1[11];	// CmdFaultReset
      S     #CmdFaultReset;
      A     "SYS_DirectCtrlDB".PC.Cmd1[13];	// CmdManualOn
      S     #InManual;
      A     "SYS_DirectCtrlDB".PC.Cmd1[14];	// CmdReportOn
      S     #InReport;
      A     "SYS_DirectCtrlDB".PC.Cmd2[13];	// CmdManualOff
      R     #InManual;
      A     "SYS_DirectCtrlDB".PC.Cmd2[14];	// CmdReportOff
      R     #InReport;
      JU    pIni;
pExa: TAR2;	// Address Dynamic datas
      T     "SYS_DirectCtrlDB".GC.InDynAddr;	// -->PCControl.GC.InDynAddr
      L     #tmpLenDyn;	// Length Dynamic datas
      T     "SYS_DirectCtrlDB".GC.InDynLen;	// -->PCControl.GC.InDynLen
      L     0;
      T     "SYS_DirectCtrlDB".GC.InParaAddr;	// -->PCControl.GC.InParaAddr
      T     "SYS_DirectCtrlDB".GC.InParaLen;	// -->PCControl.GC.InParaLen
      L     1;	// Code FcExamine
      UC    "SYS_DirectCtrl";
      L     10;	//Revision [4.2]
      T     "SYS_DirectCtrlDB".GC.Revision;
Ctrl: NOP   0;
NETWORK
TITLE =  Read from Queue (****Opto22 ****)
////*************************************************
////***             O P T O 22                    ***
////*************************************************
//
      AN    #tmpOpto22;
      JC    Ct00;
      OPN   DB [#tmpComDB];
      L     #Par.ParLCIdx;
      T     DBW 34;	//COM.Element.Index;
      L     1;	//Read LC data
      T     DBW 0;	//COM.CODE;
      CDB;
      UC    "GCS7_RS485Ctrl";
      CDB;
      L     #tmpFBNO;
      T     DBW 52;	//COM.LC0.FBNO;   
      L     DINO;
      T     DBW 54;	//COM.LC0.DINO;
      TAR2  DBD 56;	//COM.LC0.AddrDyn;        
      L     #Par.ParObjectNo;
      T     DBD 60;	//COM.LC0.AddrPara;       
      L     #Par.ParLCAddr;
      T     DBD 64;	//COM.Telegram.LCAddr;
Ct00: NOP   0;
NETWORK
TITLE =  All State Init
//===Global Group Orders===
      A     "GCS7_Gr_OutManualOn";	//Global.OutManualOn
      S     #InManual;
      A     "GCS7_Gr_OutManualOff";	//Global.OutManualOff
      R     #InManual;
      A     #InManual;
      S     "GCS7_Gr_InManual";	//Global.InManualMode
      AN    #InManual;
      A     #InLocal;
      =     #tmpLocalFault;
      A     #tmpLocalFault;
      O     #InHWStop;
      O     #InDPFault;
      =     #tmpLocal;
//---CmdFaultReset---                   //[4.9]
      A     "GCS7_Gr_OutFaultReset";	//[4.9]
      S     #CmdFaultReset;	//[4.9]
//---Report is on---
      O     "GCS7_Gr_OutReportAll";	//---Global OutReportAll
      O     #InReport;
      =     #tmpReport;
//---Enable---
      AN    #tmpLocal;
      A     #InEnable;
      AN    #CmdOff;
      =     #tmpEnable;
      AN    #tmpEnable;
      R     #OutEnabled;
//--- Fault   
      O     #OutComFault;
      AN    #tmpLocal;
      =     #tmpFault;
NETWORK
TITLE = Command to OPTO22 or commad from OTPO22
////*************************************************
////***             O P T O 22                    ***
////*************************************************
//
      AN    #tmpOpto22;
      JC    co00;
//--------------
      A     #CmdNewJob;
      AN    #Par.OutHelpFlags.CmdNewJob;
      S     #Par.OutHelpFlags.CmdNewJob;
      R     #CmdNewJob;
      A     #CmdNewValue;
      AN    #Par.OutHelpFlags.CmdNewValue;
      S     #Par.OutHelpFlags.CmdNewValue;
      R     #CmdNewValue;
//-----------------------
//New job MDEF1
      AN    #Par.ParMDEF;
      JC    co01;
      L     #Par.ParNoOfMDEF;
      L     1;
      ==I;
      A     #Par.OutHelpFlags.CmdNewJob;
      AN    #MDEF1.CmdNewRecipe;
      S     #MDEF1.CmdNewRecipe;
      R     #Par.OutHelpFlags.CmdNewJob;
//--------------
//CmdFaultReset
co01: A     #CmdFaultReset;
      S     #MYRA.Command.AlarmReset;
//--------------
//MDEF1
//--------------
      A     #MDEF1.CmdNewRecipe;
      R     #MDEF1.OutSendRecipeNrDone;
      A     #CmdFaultReset;
      S     #MDEF1.CmdAlarmReset;
      A     #MDEF1.OutWrongRecipe;
      O     #MDEF1.OutAlarm;
      O     #OutComFault;
      =     #MDEF1.StFault;
      A     #MDEF1.OutSendRecipeNrDone;
      AN    #MDEF1.StFault;
      =     #MDEF1.StOK;
      AN    #MDEF1.StOK;
      AN    #MDEF1.StFault;
      =     #MDEF1.StNotOK;
//--------------
//MDEF2
//--------------
      L     #Par.ParNoOfMDEF;	// [4.10]
      L     2;	// [4.10]
      <I;	// [4.10]
      JC    MDF3;	// [4.10]
      A     #MDEF2.CmdNewRecipe;
      R     #MDEF2.OutSendRecipeNrDone;
      A     #CmdFaultReset;
      S     #MDEF2.CmdAlarmReset;
      A     #MDEF2.OutWrongRecipe;
      O     #MDEF2.OutAlarm;
      O     #OutComFault;
      =     #MDEF2.StFault;
      A     #MDEF2.OutSendRecipeNrDone;
      AN    #MDEF2.StFault;
      =     #MDEF2.StOK;
      AN    #MDEF2.StOK;
      AN    #MDEF2.StFault;
      =     #MDEF2.StNotOK;
//--------------
//MDEF3
//--------------
MDF3: L     #Par.ParNoOfMDEF;	// [4.10]
      L     3;	// [4.10]
      <I;	// [4.10]
      JC    MDF4;	// [4.10]
      A     #MDEF3.CmdNewRecipe;
      R     #MDEF3.OutSendRecipeNrDone;
      A     #CmdFaultReset;
      S     #MDEF3.CmdAlarmReset;
      A     #MDEF3.OutWrongRecipe;
      O     #MDEF3.OutAlarm;
      O     #OutComFault;
      =     #MDEF3.StFault;
      A     #MDEF3.OutSendRecipeNrDone;
      AN    #MDEF3.StFault;
      =     #MDEF3.StOK;
      AN    #MDEF3.StOK;
      AN    #MDEF3.StFault;
      =     #MDEF3.StNotOK;
//--------------
//MDEF4
//--------------
MDF4: L     #Par.ParNoOfMDEF;	// [4.10]
      L     4;	// [4.10]
      <I;	// [4.10]
      JC    MDF5;	// [4.10]
      A     #MDEF4.CmdNewRecipe;
      R     #MDEF4.OutSendRecipeNrDone;
      A     #CmdFaultReset;
      S     #MDEF4.CmdAlarmReset;
      A     #MDEF4.OutWrongRecipe;
      O     #MDEF4.OutAlarm;
      O     #OutComFault;
      =     #MDEF4.StFault;
      A     #MDEF4.OutSendRecipeNrDone;
      AN    #MDEF4.StFault;
      =     #MDEF4.StOK;
      AN    #MDEF4.StOK;
      AN    #MDEF4.StFault;
      =     #MDEF4.StNotOK;
MDF5: NOP   0;
//--------------
//MYRA
//--------------
      A     #OutpRelease;
      A     #Par.ParMYRA;
      =     #MYRA.Command.Start;
//--------------
//MYAG
//--------------
      A     #OutpRelease;
      A     #Par.ParMYAG;
      =     #MYAG.Start;
//--------------
//Alarms
//Copy alarm from OPTO2 to digital inputs signal 
//--------------
      NOP   0;	//----MYRA------------
      A     #MYRA.OutAlarm.AlarmMYRAHardware;
      O     #MYRA.OutAlarm.AlarmFeeder1;
      O     #MYRA.OutAlarm.AlarmFeeder2;
      O     #MYRA.OutAlarm.AlarmFeeder3;
      O     #MYRA.OutAlarm.AlarmFeeder4;
      A     #Par.ParMYRA;
      O;	//----MYAG------------
      A     #MYAG.OutSumFault;
      A     #Par.ParMYAG;
      O;	//----MDEF------------
      A(;
      L     #Par.ParNoOfMDEF;
      L     1;
      ==I;
      A     #Par.ParMDEF;
      A     #MDEF1.OutAlarm;
      );
      =     #InpFaultLc;
//======================================
//Tolerance alarm
      A     #MYRA.OutAlarm.AlarmProduct;
      A     #Par.ParMYRA;
      =     #InpOutOfTolerance;
//===============================================
//Definition fault
      NOP   0;	//----MYRA-----------
      A     #MYRA.OutAlarm.AlarmRecipeChange;
      A     #Par.ParMYRA;
      O;	//----MDEF------------
      A(;
      L     #Par.ParNoOfMDEF;
      L     1;
      ==I;
      A     #Par.ParMDEF;
      A     #MDEF1.OutWrongRecipe;
      );
      =     #InDefFault;
//Definiton ready
      NOP   0;	//----MYAG-----------
      L     #MYAG.OutRecipeNr;
      L     #MYAG.InRecipeNr;
      ==D;
      A(;
      L     #MYAG.InJobNr;
      L     #MYAG.OutJobNr;
      ==D;
      );
      A     #Par.ParMYAG;
      O;	//----MYRA-----------
      AN    #Par.OutHelpFlags.CmdNewJob;
      A     #Par.ParMYRA;
      AN    #InDefFault;
      O;	//----MDEF------------
      A(;
      L     #Par.ParNoOfMDEF;
      L     1;
      <>I;
      ON    #MDEF1.CmdNewRecipe;
      );
      AN    #InDefFault;
      A     #Par.ParMDEF;
      =     #InDefReady;
co00: NOP   0;
NETWORK
TITLE = States
//===State machine===
      A     #StOff;
      JC    S0;
      A     #StOn;
      JC    S2;
      A     #StWaitForResponse;
      JC    S1;
      A     #StCtoFault;
      JC    S3;
      A     #StFault;
      JC    S4;
      S     #StOff;	// Init
NETWORK
TITLE = StOff
// Any transition to StOff
xxS0: S     #StOff;
      R     #OutpAlarmReset;
      R     #OutEnabled;
      JU    LOGx;
//=== Logic ====
//Transition to StOn
S0:   A(;
      A     #CmdNext;
      AN    #InManual;
      O     #CmdOn;
      O;
      A     #MYRA.OutStatus.Started;
      A     #Par.ParMYRA;
      );
      A     #tmpEnable;
      AN    #tmpLocal;
      R     #StOff;
      JC    xxS2;
//Transition to StFault
      A     #tmpFault;
      AN    #InNoMonLC;	//[4.5]
      R     #StOff;
      R     #OutWarning;
      JC    xxS4;	//-->StFault
//Transition to StWaitForResponse 
      AN    #InDefReady;
      AN    #tmpLocal;
      R     #StOff;
      JC    xxS1;
      JU    LOG4;
NETWORK
TITLE = StWaitForResponse
// Any transition to StOn
xxS1: S     #StWaitForResponse;
      L     #Par.ParResponseTime;
      T     #Par.OutDelayTime;
//=== Logic ====
S1:   AN    "GCS7_Gr_OutTick200ms";	//Gr.OutTick200ms
      L     #Par.OutDelayTime;
      JC    S1J3;
      +     -2;
      T     #Par.OutDelayTime;
S1J3: L     0;
      <=I;
      =     #tmpTimeDone;
//Transition to StOff
      A     #InDefReady;
      AN    #OutEnabled;	//[4.4] 
      AN    #OutpAlarmReset;
      O     #tmpLocal;
      R     #StWaitForResponse;
      JC    xxS0;	//-->StOff                
//Transition to StFault 
      A     #InDefFault;
      O     #tmpTimeDone;
      O     #tmpFault;
      AN    #InNoMonLC;	//[4.5]
      R     #StWaitForResponse;
      JC    xxS4;
//Transition to StOn
      A     #InDefReady;
      A     #OutEnabled;
      O     #InNoMonLC;	//[4.5]
      R     #StWaitForResponse;
      JC    xxS2;	//-->StOn         
      JU    LOG4;
NETWORK
TITLE = StOn
// Any transition to StOn
xxS2: S     #StOn;
      R     #OutpAlarmReset;
      S     #OutEnabled;
      L     #Par.ParDelayWarning;
      T     #Par.OutDelayTime;
      JU    LOGx;
//=== Logic ====
S2:   A     #InpFaultLc;	//[4.3]
      A     #InNoMonLC;	//[4.3]
      O     #InpOutOfTolerance;
      JC    S2J1;
      R     #OutWarning;
      L     #Par.ParDelayWarning;
      T     #Par.OutDelayTime;
      JU    S2J2;
//Delay time warning
S2J1: A     #OutWarning;
      JC    S2J2;
      AN    "GCS7_Gr_OutTick200ms";	//Gr.OutTick200ms
      L     #Par.OutDelayTime;
      JC    S2J3;
      +     -2;
      T     #Par.OutDelayTime;
S2J3: L     0;
      <=I;
      S     #OutWarning;
//Transition to StOff
S2J2: AN    #tmpEnable;
      R     #StOn;
      R     #OutWarning;
      JC    xxS0;	//-->StOff
//Transition to StWaitForResponse
      A     #OutDefRequested;
      R     #StOn;
      R     #OutWarning;
      JC    xxS1;	//-->StWaitForResponse
//Transition to StFault
      A     #InDefFault;
      O     #tmpFault;
      AN    #InNoMonLC;	//[4.5]
      R     #StOn;
      R     #OutWarning;
      JC    xxS4;	//-->StFault
//Transition to StCtoFault
      A     #OutWarning;
      A     #Par.ParMDEx;
      O     #InpFaultLc;
      AN    #InNoMonLC;	//[4.3]
      R     #StOn;
      R     #OutWarning;
      JC    xxS3;	//-->StCtoFault
      JU    LOG4;
NETWORK
TITLE = StCtoFault
// Any transition to StOn
xxS3: S     #StCtoFault;
      L     #Par.ParDelayFault;
      T     #Par.OutDelayTime;
//=== Logic ====
S3:   AN    "GCS7_Gr_OutTick200ms";	//Gr.OutTick200ms
      L     #Par.OutDelayTime;
      JC    S3J3;
      +     -2;
      T     #Par.OutDelayTime;
S3J3: L     0;
      <=I;
      =     #tmpTimeDone;
//Transition to StFault
      A     #InDefFault;
      O     #tmpTimeDone;
      O     #tmpFault;
      R     #StCtoFault;
      JC    xxS4;	//-->StFault
//Transition to StWaitForResponse
      A     #OutDefRequested;
      R     #StCtoFault;
      JC    xxS1;	//-->StWaitForResponse
//Transition to StOff
      AN    #tmpEnable;
      R     #StCtoFault;
      JC    xxS0;	//-->StOff
//Transition to StOn
      AN    #Par.ParMDEx;
      ON    #InpOutOfTolerance;
      AN    #InpFaultLc;
      R     #StCtoFault;
      JC    xxS2;	//-->StOn
      JU    LOG4;
NETWORK
TITLE = StFault
// Any transiton to Fault  
xxS4: S     "GCS7_Gr_InFaultFlag";	//Gr.InFaultFlag
      S     #StFault;
      R     #OutpAlarmReset;
      R     #Par.OutHelpFlags.OutTestNewAlarm;
      R     #Par.OutHelpFlags.OutFaultResetDone;
      CALL  "SYS_Horn_Code" (
           FcCode                   := 1,
           ParObjectType            := 1036,
           ParObjectNo              := #Par.ParObjectNo,
           ParHornCode              := #Par.ParHornCode);
      L     #Par.ParAlarmResetTime;
      T     #Par.OutDelayTime;
      JU    LOG4;
//=== Logic ====
S4:   AN    "GCS7_Gr_OutTick200ms";	//Gr.OutTick200ms
      ON    #OutpAlarmReset;
      L     #Par.OutDelayTime;
      JC    S4J3;
      +     -2;
      T     #Par.OutDelayTime;
S4J3: L     0;
      <I;	//[4.1]
      =     #tmpTimeDone;
//Send command to MYRA
      A     #CmdFaultReset;
//[4.9]      O     M     12.3                  //Gr.OutFaultReset
      S     #OutpAlarmReset;
//Transition to StOn                      [4.6]
      AN    #tmpFault;	//[4.6]
      A     #InNoMonLC;	//[4.6]
      R     #StFault;	//[4.6]
      S     #StOn;	//[4.6]
      R     #OutpAlarmReset;	//[4.6]
      JC    LOGC;	//--> StOn   [4.6]
//Transition to StOff
      A     #OutpAlarmReset;
      AN    #InDefFault;
      AN    #InpFaultLc;
      AN    #tmpFault;
      O     #InNoMonLC;	//[4.5]
      O     #tmpLocalFault;
      R     #StFault;
      S     #StOff;
      R     #OutpAlarmReset;
      JC    LOGC;	//--> StOff       
//Retry fault
      A     #Par.ParMYRA;
      O     #Par.ParMDEF;
      A     #Par.OutHelpFlags.OutTestNewAlarm;
      O;
      AN    #Par.ParMYRA;
      AN    #Par.ParMDEF;
      A     #OutpAlarmReset;
      A     #tmpTimeDone;
      JC    S4J1;
//[5.0]      JU    LOG4
      JU    OUT;	//[5.0]
//Check new alarms
//Clear Par.OutMsg
S4J1: L     0;
      T     DID [#tmpAddrMsg];
      JC    xxS4;
NETWORK
TITLE = LOG
LOGx: L     B#(4, 0);	// Message ('Off')
      A     #StOff;
      A     #InReport;
      JC    LOG;
      L     B#(4, 1);	// Message ('On')
      A     #StOn;
      A     #InReport;
      JC    LOG;
      JU    OUT;
//--------------
//Check new MDEF alarm
LOG4: A     #tmpLocal;
      JC    OUT;
      AN    #Par.ParMDEF;
      JC    LOG5;
      A     #MDEF1.OutAlarm;
      FP    #OutMsg.A41Mill1;
      L     B#(4, 41);	// Message ('Alarm MDEF mill 1' )
      JC    LOG;
      A     #MDEF2.OutAlarm;
      FP    #OutMsg.A42Mill2;
      L     B#(4, 42);	// Message ('Alarm MDEF mill 2' )
      JC    LOG;
      A     #MDEF3.OutAlarm;
      FP    #OutMsg.A43Mill3;
      L     B#(4, 43);	// Message ('Alarm MDEF mill 3' )
      JC    LOG;
      A     #MDEF4.OutAlarm;
      FP    #OutMsg.A44Mill4;
      L     B#(4, 44);	// Message ('Alarm MDEF mill 4' )
      JC    LOG;
      A     #MDEF1.OutWrongRecipe;
      FP    #OutMsg.A51RecipeMill1;
      L     B#(4, 51);	// Message ('Alarm recipe MDEF mill 1' )
      JC    LOG;
      A     #MDEF2.OutWrongRecipe;
      FP    #OutMsg.A52RecipeMill3;
      L     B#(4, 52);	// Message ('Alarm recipe MDEF mill 2' )
      JC    LOG;
      A     #MDEF3.OutWrongRecipe;
      FP    #OutMsg.A53RecipeMill2;
      L     B#(4, 53);	// Message ('Alarm recipe MDEF mill 3' )
      JC    LOG;
      A     #MDEF4.OutWrongRecipe;
      FP    #OutMsg.A54RecipeMill4;
      L     B#(4, 54);	// Message ('Alarm recipe MDEF mill 4' )
      JC    LOG;
//----------------
//Check new MYRA alarm
LOG5: AN    #Par.ParMYRA;
      JC    LOG6;
      L     B#(4, 21);	// Message ('MYRA Alarm hardware' )
      A     #MYRA.OutAlarm.AlarmMYRAHardware;
      A     #StFault;
      FP    #OutMsg.A21MYRAHardware;
      JC    LOG;
      L     B#(4, 22);	// Message ('MYRA Alarm product' )
      A     #MYRA.OutAlarm.AlarmProduct;
      A     #StFault;
      FP    #OutMsg.A22MYRAProduct;
      JC    LOG;
      L     B#(4, 23);	// Message ('MYRA RecipeChange' )
      A     #MYRA.OutAlarm.AlarmRecipeChange;
      A     #StFault;
      FP    #OutMsg.A23MYRARecipeChange;
      JC    LOG;
      A     #MYRA.OutAlarm.AlarmFeeder1;
      A     #StFault;
      L     B#(4, 24);	// Message ('MYRA Feeder1' )
      FP    #OutMsg.A24MYRAFeeder1;
      JC    LOG;
      A     #MYRA.OutAlarm.AlarmFeeder2;
      A     #StFault;
      L     B#(4, 25);	// Message ('MYRA Feeder2' )
      FP    #OutMsg.A25MYRAFeeder2;
      JC    LOG;
      A     #MYRA.OutAlarm.AlarmFeeder3;
      A     #StFault;
      L     B#(4, 26);	// Message ('MYRA Feeder3' )
      FP    #OutMsg.A26MYRAFeeder3;
      JC    LOG;
      A     #MYRA.OutAlarm.AlarmFeeder4;
      A     #StFault;
      L     B#(4, 27);	// Message ('MYRA Feeder4' )
      FP    #OutMsg.A27MYRAFeeder4;
      JC    LOG;
//----------------
//Check new ALL
LOG6: L     B#(4, 15);	// Message ('fault communication OPTO22' )
      A     #OutComFault;
      A     #StFault;
      FP    #OutMsg.A15CommunicationLC;
      JC    LOG;
      A     #InDefFault;
      ON    #InDefReady;
      A     #StFault;
      L     B#(4, 12);	// Message ('fault transmision' )
      FP    #OutMsg.A12CommunicationPC;
      JC    LOG;
      A     #InpOutOfTolerance;
      A     #StFault;
      L     B#(4, 11);	// Message ('fault tolerance' ) 
      FP    #OutMsg.A11Tolerance;
      JC    LOG;
      L     B#(1, 10);	// Message ('fault equipement' )
      A     #InpFaultLc;
      A     #StFault;
      FP    #OutMsg.A10LC;
      JC    LOG;
      JU    OUT;
LOGC: L     B#(3, 9);	//Message ('fault cancelled')
LOG:  A     #Par.ParLogOff;	//---Set LOG Message
      JC    OUT;
      T     #tmpLOGvalue;
      L     W#16#FF;
      AW;
      T     #OutAlarmNrLog;
      CALL  "GCS7_LogConvert" (
           ObjectNo                 := #Par.ParObjectNo,
           MsgType                  := #Par.ParMsgType,
           ClassMsgTxt              := #tmpLOGvalue,
           OType                    := 1036);	// LOG Message Converter / Entry / Contains Class and TextNo
//===================================================================
//Clear Alarm Nr
OUT:  L     0;
      L     DID [#tmpAddrMsg];	//OutMsg
      <>D;
      =     #Par.OutHelpFlags.OutAlarmActive;
      L     10;
      L     #OutAlarmNrLog;
      <=I;
      AN    #Par.OutHelpFlags.OutAlarmActive;
      AN    #StFault;
      JCN   OUT2;
      L     0;
      T     #OutAlarmNrLog;
OUT2: NOP   0;
NETWORK
TITLE = Global End
      CLR;	//---Clear all commands
      =     #CmdOn;
      =     #CmdOff;
      =     #CmdNext;
      =     #CmdFaultReset;
      AN    #tmpLocal;
      A     #OutEnabled;
      =     #OutpRelease;
      AN    #tmpLocal;
      AN    #InDefReady;
      =     #OutDefRequested;
//--Output for group 
      A     #InDPFault;
      AN    #tmpLocalFault;
      S     "GCS7_Gr_InDPFault";
      A     #InHWStop;
      AN    #tmpLocalFault;
      S     "GCS7_Gr_InHWStop";
NETWORK
TITLE = State Code
      AN    #StOff;
      JC    STC2;
      L     41;	//Code: StOff.HWStop
      A     #InHWStop;
      JC    STC9;
      L     51;	//Code: StOff.DPFault
      A     #InDPFault;
      JC    STC9;
      L     1;	//Code: StOff
      JU    STC9;
STC2: A     #StWaitForResponse;
      L     2;	// Code: StWaitForResponse
      JC    STC9;
      A     #StOn;
      AN    #OutWarning;
      L     3;	// Code: StOn.Ok
      JC    STC9;
      A     #StOn;
      L     4;	// Code: StOn.Warning
      JC    STC9;
      A     #StCtoFault;
      L     5;	// Code: StCtoFault
      JC    STC9;
      L     32;	// Code: fault
STC9: L     #StCode;	// Old state code
      TAK;
      T     #StCode;	// Save state code
      <>I;
      L     3;	// Load code for CBit methode
      CC    "SYS_CBitCtrl";
NETWORK
TITLE = Communication
////*************************************************
////***             O P T O 22                    ***
////*************************************************
//
      AN    #tmpOpto22;
      JC    com0;
      A     DBX 50.0;	//COM.LC0.CmdPut
      O     DBX 50.1;	//COM.LC0.CmdGet
      JC    com0;
//--- 'I'
      AN    #Par.OutComFlags.I_Done;
      A     #Par.ParMYAG;
      L     'I';
      JC    PUT;
//--- 'b' MYAG
      AN    #Par.OutComFlags.b_Done;
      A     #Par.ParMYAG;
      S     #Par.OutComFlags.b_Done;
      L     'b';
      JC    GET;
//[5.2]--- 'b' MYRA
      AN    #Par.OutComFlags.b_Done;	//[5.2]
      A     #Par.ParMYRA;	//[5.2]
      S     #Par.OutComFlags.b_Done;	//[5.2]
      L     'b';	//[5.2]
      JC    GET;	//[5.2]
//[5.2] --- 'N'
      AN    #Par.OutComFlags.N_Done;	//[5.2] 
      A     #Par.ParMYRA;	//[5.2] 
      S     #Par.OutComFlags.N_Done;	//[5.2] 
      L     'N';	//[5.2] 
      JC    PUT;	//[5.2] 
//[5.0] --- 'm'
      AN    #Par.OutComFlags.m_Done;	//[5.0] 
      A     #Par.ParMYRA;	//[5.0] 
      S     #Par.OutComFlags.m_Done;	//[5.0] 
      L     'm';	//[5.0] 
      JC    PUT;	//[5.0] 
//--- 'P'
      AN    #Par.OutComFlags.P_Done;
      A     #Par.OutHelpFlags.CmdNewJob;
      A     #Par.ParMYRA;
      L     'P';
      JC    PUT;
//--- 'Q'
      AN    #Par.OutComFlags.Q_Done;
      A     #Par.OutHelpFlags.CmdNewValue;
      A     #Par.ParMYRA;
      L     'Q';
      JC    PUT;
//--- 'S'
      A(;
      A     #MYRA.Command.Start;
      AN    #MYRA.OutStatus.Started;
      AN    #MYRA.OutStatus.Suspended;	//[4.7]
      AN    #MYRA.OutAlarm.AlarmMYRAHardware;
      O(;
      A     #MYRA.OutStatus.Started;
      O     #MYRA.OutStatus.Suspended;	//[4.7]
      AN    #MYRA.Command.Start;
      );
      O;
      X     #MYRA.Command.CheckLimit;
      X     #Par.OutHelpFlags.FlagCheckLimit;
      O     #MYRA.Command.AlarmReset;
      );
      AN    #Par.OutComFlags.S_Done;
      A     #Par.ParMYRA;
      L     'S';
      JC    PUT;
//--- 'a'
      AN    #Par.OutComFlags.a_rDone;
      A     #Par.ParMYRA;
      S     #Par.OutComFlags.a_rDone;
      L     'a';
      JC    GET;
//--- 'f'                     //[4.0]
      AN    #Par.OutComFlags.f_rDone;	//[4.0]
      A     #Par.ParMYRA;	//[4.0]
      S     #Par.OutComFlags.f_rDone;	//[4.0]
      L     'f';	//[4.0]
      JC    GET;	//[4.0]
//--- 'i'                     //[5.1]
      AN    #Par.OutComFlags.i_rDone;	//[5.1]
      A     #Par.ParMYRA;	//[5.1]
      S     #Par.OutComFlags.i_rDone;	//[5.1]
      L     'i';	//[5.1]
      JC    GET;	//[5.1]
//--- 's'
      AN    #Par.OutComFlags.s_rDone;
      A     #Par.ParMYRA;
      S     #Par.OutComFlags.s_rDone;
      L     's';
      JC    GET;
      AN    #Par.ParMDEF;
      JC    oA0;
// Mill 1
//--- 'D'
      AN    #Par.OutComFlags.D_Done;
      A     #MDEF1.CmdNewRecipe;
      AN    #MDEF1.OutSendRecipeNrActive;	//[4.8]
      AN    #MDEF2.OutSendRecipeNrActive;	//[4.8]
      AN    #MDEF3.OutSendRecipeNrActive;	//[4.8]
      AN    #MDEF4.OutSendRecipeNrActive;	//[4.8]
      A     #Par.ParMDEF;
      JCN   oA1;
      L     1;
      T     #Par.OutMillNr;
      L     'D';
      JU    PUT;
//--- 'A'
oA1:  AN    #Par.OutComFlags.A_Done;
      A     #MDEF1.CmdAlarmReset;
      A     #Par.ParMDEF;
      JCN   oD2;
      R     #MDEF1.CmdAlarmReset;
      L     1;
      T     #Par.OutMillNr;
      L     'A';
      JU    PUT;
// Mill 2
//--- 'D'
oD2:  AN    #Par.OutComFlags.D_Done;
      A     #MDEF2.CmdNewRecipe;
      AN    #MDEF1.OutSendRecipeNrActive;	//[4.8]
      AN    #MDEF2.OutSendRecipeNrActive;	//[4.8]
      AN    #MDEF3.OutSendRecipeNrActive;	//[4.8]
      AN    #MDEF4.OutSendRecipeNrActive;	//[4.8]
      A     #Par.ParMDEF;
      JCN   oA2;
      L     2;
      T     #Par.OutMillNr;
      L     'D';
      JU    PUT;
//--- 'A'
oA2:  AN    #Par.OutComFlags.A_Done;
      A     #MDEF2.CmdAlarmReset;
      A     #Par.ParMDEF;
      JCN   oD3;
      R     #MDEF2.CmdAlarmReset;
      L     2;
      T     #Par.OutMillNr;
      L     'A';
      JU    PUT;
// Mill 3
//--- 'D'
oD3:  AN    #Par.OutComFlags.D_Done;
      A     #MDEF3.CmdNewRecipe;
      AN    #MDEF1.OutSendRecipeNrActive;	//[4.8]
      AN    #MDEF2.OutSendRecipeNrActive;	//[4.8]
      AN    #MDEF3.OutSendRecipeNrActive;	//[4.8]
      AN    #MDEF4.OutSendRecipeNrActive;	//[4.8]
      A     #Par.ParMDEF;
      JCN   oA3;
      L     3;
      T     #Par.OutMillNr;
      L     'D';
      JU    PUT;
//--- 'A'
oA3:  AN    #Par.OutComFlags.A_Done;
      A     #MDEF3.CmdAlarmReset;
      A     #Par.ParMDEF;
      JCN   oD4;
      R     #MDEF3.CmdAlarmReset;
      L     3;
      T     #Par.OutMillNr;
      L     'A';
      JU    PUT;
// Mill 4
//--- 'D'
oD4:  AN    #Par.OutComFlags.D_Done;
      A     #MDEF4.CmdNewRecipe;
      AN    #MDEF1.OutSendRecipeNrActive;	//[4.8]
      AN    #MDEF2.OutSendRecipeNrActive;	//[4.8]
      AN    #MDEF3.OutSendRecipeNrActive;	//[4.8]
      AN    #MDEF4.OutSendRecipeNrActive;	//[4.8]
      A     #Par.ParMDEF;
      JCN   oA4;
      L     4;
      T     #Par.OutMillNr;
      L     'D';
      JU    PUT;
//--- 'A'
oA4:  AN    #Par.OutComFlags.A_Done;
      A     #MDEF4.CmdAlarmReset;
      A     #Par.ParMDEF;
      JCN   oA0;
      R     #MDEF4.CmdAlarmReset;
      L     4;
      T     #Par.OutMillNr;
      L     'A';
      JU    PUT;
oA0:  NOP   0;
//--- 's'
      A     #MDEF1.OutSendRecipeNrActive;	//[4.8]
      O     #MDEF2.OutSendRecipeNrActive;	//[4.8]
      O     #MDEF3.OutSendRecipeNrActive;	//[4.8]
      O     #MDEF4.OutSendRecipeNrActive;	//[4.8]
      AN    #Par.OutComFlags.s_rDone;
      A     #Par.ParMDEF;
      S     #Par.OutComFlags.s_rDone;
      L     's';
      JC    GET;
//--- 'a'
      AN    #Par.OutComFlags.a_rDone;
      A     #Par.ParMDEF;
      S     #Par.OutComFlags.a_rDone;
      L     'a';
      JC    GET;
      JU    CmCR;
PUT:  SET;
      S     DBX 50.0;	//COM.LC0.CmdPut ;
      T     DBB 51;	//COM.LC0.Command;
      JU    com0;
GET:  SET;
      S     DBX 50.1;	//COM.LC0.CmdGet ;
      T     DBB 51;	//COM.LC0.Command;
      JU    com0;
// 
//---Clear command flags (x_done)
CmCR: SET;
      R     #Par.OutComFlags.a_rDone;
      R     #Par.OutComFlags.s_rDone;
      R     #Par.OutComFlags.k_Done;
      R     #Par.OutComFlags.b_Done;
      R     #Par.OutComFlags.D_Done;
      R     #Par.OutComFlags.A_Done;
      R     #Par.OutComFlags.P_Done;
      R     #Par.OutComFlags.Q_Done;
      R     #Par.OutComFlags.S_Done;
      R     #Par.OutComFlags.I_Done;
      R     #Par.OutComFlags.f_rDone;	//[4.0]
      R     #Par.OutComFlags.m_Done;	//[5.0]
      R     #Par.OutComFlags.i_rDone;	//[5.1]
      R     #Par.OutComFlags.N_Done;	//[5.2]
com0: NOP   0;
NETWORK
TITLE =  Store LC data (***OPTO22 **)
////*************************************************
////***             O P T O 22                    ***
////*************************************************
//
      AN    #tmpOpto22;
      BEC;
      L     #Par.ParLCIdx;
      T     DBW 34;	//COM.Element.Index; 
      L     2;	//Store LC data
      T     DBW 0;	//COM.CODE;
      CDB;
      UC    "GCS7_RS485Ctrl";
      CDB;
      BEU;
END_FUNCTION_BLOCK

